PROGRAM MAIN

// MOTOR WITH LIGHT AND BUTTON BRANCH

VAR
	motor : FB_XenaxAxisForceFeedback;
	motorSequence : ST_MOTION_PARAMS;
	
	initialSetup : BOOL := TRUE;
	
	justAStep : BOOL := TRUE;
	
	
	enumStates : (INITIALIZE_VALUES, INITIALIZE, FETCH, MOVING, WAIT, GET_NEXT_TARGET, MOVE_TO_TARGET);
	
	aTargets : ARRAY[1..10] OF INT := [0, 360, 720, 0, 720, -720, 0, -360, 360, 0];
	nTargetIndex : INT := 1;
	nTargetValue : INT := 0;
	
	tonWaitTimer : TON := (PT := T#500MS);
	
	// could do array to track state number, better for scalability
	//aMoveState : ARRAY[1..4] OF enumStates := [=(MOVE1, MOVE2, MOVE3, MOVE4);
	//nMoveState : INT := 1;
	dbg : INT;
	
	
END_VAR

motor(usiRefernceDirection := INT_TO_USINT(E_JS_MC_REF_MODE.Positive));

CASE enumStates OF
	INITIALIZE_VALUES:
		motorSequence.TargetPos := 0;
		motorSequence.Jerk := 20000;
		motorSequence.TargetAccel := 2000;
		motorSequence.TargetDecel := 2000;
		motorSequence.TargetVel := 1000;
		enumStates := INITIALIZE;
		
	INITIALIZE:
		motor.Initialize(TRUE);
		IF motor.DidInitialize THEN
			nTargetValue := 0;
			enumStates := MOVE_TO_TARGET;
		END_IF
		
	MOVING:
		motor.MoveAbs(Execute := TRUE, MotionParams := motorSequence);
		IF motor.DidMoveAbs THEN
			motor.MoveAbs(Execute := FALSE, MotionParams := motorSequence);
			enumStates := WAIT;
		END_IF
		
	WAIT:
		tonWaitTimer(IN := TRUE);
		
		IF tonWaitTimer.Q THEN
			tonWaitTimer(IN := FALSE);
			enumStates := GET_NEXT_TARGET;
		END_IF
		// wait code here
		// if time elapsed then go to next state
		// after waiting the duration the if statement is triggered
		// inside the if statement can increment the moveState variable
		
		//enumStates := GET_NEXT_TARGET;
		
	GET_NEXT_TARGET:
		dbg := UINT_TO_INT(SIZEOF(aTargets)/2); // divide by 2 since the array type is of int (2 bytes per entry)
		IF nTargetIndex + 1 > UINT_TO_INT(SIZEOF(aTargets)/2) THEN // divide by 2 since the array type is of int (2 bytes per entry)
			nTargetIndex := 1;
		END_IF

		nTargetValue := aTargets[nTargetIndex];
		
		nTargetIndex := nTargetIndex + 1;
		
		enumStates := MOVE_TO_TARGET;
		
	
		
	MOVE_TO_TARGET:
		motorSequence.TargetPos := nTargetValue;
		enumStates := MOVING;
	
		
END_CASE


(*
IF initialSetup THEN
	motor.Initialize(TRUE);
	motorSequence.TargetPos := 10000;
	//motorSequence.TargetDistance := 50000;
	motorSequence.Jerk := 20000;
	motorSequence.TargetAccel := 2000;
	motorSequence.TargetDecel := 2000;
	motorSequence.TargetVel := 1000;
	
	IF motor.DidInitialize THEN
			initialSetup := FALSE;
	END_IF

ELSE
	motor.MoveAbs(Execute := TRUE, MotionParams := motorSequence);

	IF motor.DidMoveAbs THEN
		motor.MoveAbs(Execute := FALSE, MotionParams := motorSequence);
	END_IF
	
END_IF
*)

END_PROGRAM

(* stored: Version 1.1.0.1, ProductVersion 3.1.4024.12
   POU MAIN: Id {3cca0f7b-1c22-4553-a492-10a9c50dc7a8}, SpecialFunc None *)
